{attribute 'qualified_only'}
VAR_GLOBAL
	//SafetyOK				: BOOL;
	AllChargeRelayClosed 	: BOOL := 0;
	AllDumpRelayOpen		: BOOL := 0;
	//AllDumpRelayClose		: BOOL := 0;
	ReadyToCharge			: BOOL := 0;
	AllChargerEOC			: BOOL := 0;
	
	ChargerVBelowThres		: BOOL := 0;
	ChargerVThres			: REAL := 40;
	AllChargerHVisOFF		: BOOL := 0;
	AllChargerInhibitON		: BOOL := 0;

	AllCapsDischarged		: BOOL := 0;
	CapVoltageThres			: REAL := 40;
	SystemIsSafe			: BOOL := 0;
END_VAR

(* stored: Version 1.1.0.1, ProductVersion 3.1.4024.11
   GVL Permissives_DB: Id {c05a4b99-99cd-4605-96e2-a97127a00965} *)
